// TIA Portal V20 export
// export: Created 2025-12-01T14:57:46.8015245Z, ExportSetting None, DisplayName Totally Integrated Automation Portal, DisplayVersion V20 Update 3, DisplayName TIA Portal Openness, DisplayVersion V20 Update 3, DisplayName TIA Portal Version Control Interface, DisplayVersion V20 Update 3, DisplayName STEP 7 Professional, DisplayVersion V20 Update 3, DisplayName STEP 7 Safety, DisplayVersion V20 Update 2, DisplayName WinCC Basic/Comfort/Advanced, DisplayVersion V20 Update 3, DisplayName WinCC Professional, DisplayVersion V20 Update 3, DisplayName WinCC Unified, DisplayVersion V20 Update 3
DATA_BLOCK "DB210_DB_Eventos_Router"   // DB210
{ S7_Optimized_Access := 'FALSE' }
// stored: AutoNumber false
   VAR
      EVENTO : Array[1..2600] of Char;
   END_VAR
BEGIN
END_DATA_BLOCK
